Yaskawa INFORM job: N_R2_D54(P)(-165,-90).JBI

/JOB
//NAME N_R2_D54(P)(-165,-90)
//POS
///NPOS 418,418,418,21,0,0
///TOOL 0
///POSTYPE PULSE
///PULSE
C00000=-39723,-76225,-106677,19950,71807,76871
C00001=-136716,-73683,-105524,19345,72156,77265
C00002=-161407,-91524,-110310,15012,103390,71507
C00003=-159933,-105942,-63343,4894,72862,63752
C00004=-161158,-104529,-58514,4950,70696,63247
C00005=-161668,-103884,-56534,4974,69842,63039
C00006=-161778,-102512,-54221,4996,69133,62972
C00007=-161760,-102726,-54587,4993,69247,62982
C00008=-161816,-102665,-54558,4992,69263,62964
C00009=-163044,-104500,-55207,5003,68794,62527
C00010=-161816,-102665,-54558,4992,69263,62964
C00011=-161303,-103338,-56557,4967,70114,63174
C00012=-160072,-104820,-61433,4909,72274,63681
C00013=-171279,-139675,-91122,7314,74940,61433
C00014=-160786,-120191,-86572,7704,81092,65337
C00015=-161517,-119982,-82352,7740,78693,64939
C00016=-161824,-119782,-80612,7757,77762,64776
C00017=-161934,-118571,-78477,7774,77087,64696
C00018=-161898,-118737,-78823,7771,77210,64716
C00019=-161973,-118676,-78783,7769,77224,64692
C00020=-163205,-120940,-79512,7761,76632,64235
C00021=-161973,-118676,-78783,7769,77224,64692
C00022=-161664,-118910,-80540,7751,78148,64855
C00023=-160927,-119214,-84804,7712,80524,65254
C00024=-170669,-154499,-108862,8582,79492,59623
C00025=-160866,-130175,-103256,9154,87324,63496
C00026=-161601,-130979,-99438,9146,84678,63052
C00027=-161908,-131130,-97845,9147,83668,62873
C00028=-162018,-130031,-95808,9153,82999,62786
C00029=-162011,-130213,-96119,9152,83096,62795
C00030=-162089,-130094,-96081,9149,83142,62772
C00031=-163326,-132893,-96929,9116,82375,62294
C00032=-162089,-130094,-96081,9149,83142,62772
C00033=-161779,-129993,-97692,9146,84137,62951
C00034=-161038,-129333,-101562,9150,86742,63395
C00035=-164208,-146274,-116147,-5663,80658,78475
C00036=-172457,-131111,-102504,-10822,75194,76159
C00037=-174484,-130450,-98260,-10690,72692,75663
C00038=-175320,-130052,-96514,-10635,71726,75451
C00039=-175466,-128922,-94464,-10657,71037,75460
C00040=-175415,-129062,-94788,-10656,71169,75467
C00041=-175494,-129100,-94788,-10647,71140,75441
C00042=-177063,-131522,-95540,-10496,70167,74966
C00043=-175494,-129100,-94788,-10647,71140,75441
C00044=-174655,-129535,-96550,-10701,72096,75655
C00045=-172620,-130306,-100836,-10831,74570,76157
C00046=-185476,-152836,-107470,-9889,65575,72355
C00047=-172370,-120582,-85424,-11113,70194,76647
C00048=-174396,-119219,-80852,-11015,67845,76138
C00049=-175231,-118580,-78981,-10974,66925,75923
C00050=-175377,-117338,-76830,-11009,66232,75936
C00051=-175358,-117539,-77175,-11003,66341,75932
C00052=-175389,-117510,-77167,-10998,66348,75920
C00053=-176957,-119476,-77818,-10848,65543,75427
C00054=-175389,-117510,-77167,-10998,66348,75920
C00055=-174552,-118176,-79054,-11039,67264,76137
C00056=-172519,-119613,-83665,-11134,69599,76649
C00057=-182787,-134787,-88740,-10457,63687,73508
C00058=-171653,-105129,-60487,-14223,60495,76409
C00059=-174094,-102685,-55336,-14102,58231,75776
C00060=-175092,-101639,-53233,-14049,57333,75512
C00061=-175238,-100225,-50886,-14136,56611,75552
C00062=-175227,-100493,-51313,-14118,56735,75540
C00063=-175234,-100467,-51279,-14118,56726,75538
C00064=-176798,-102054,-51863,-13921,56030,75027
C00065=-175234,-100467,-51279,-14118,56726,75538
C00066=-174232,-101534,-53401,-14169,57626,75804
C00067=-171784,-104034,-58596,-14285,59890,76439
C00068=-145436,-132678,-96384,-390,75100,72869
C00069=-145436,-153477,-122592,-390,33068,72869
C00070=-145436,-153477,-122592,-390,33068,72869
C00071=-145875,-137223,-99163,-150,44123,76557
C00072=-145875,-137223,-99163,3185,26782,75636
C00073=-145939,-91194,-32923,8725,9743,73059
C00074=-160530,-30732,15414,32644,16120,44715
C00075=-161197,-23323,24436,37351,14921,42434
C00076=-161451,-20239,28250,39583,14417,41366
C00077=-161567,-18480,31613,42866,13575,39840
C00078=-161451,-20239,28250,39583,14417,41366
C00079=-161554,-18653,31308,42567,13643,39979
C00080=-160680,-16153,33400,41106,13277,40797
C00081=-161554,-18653,31308,42567,13643,39979
C00082=-161301,-21808,27395,40043,14138,41179
C00083=-160636,-29361,18168,34773,15327,43713
C00084=-135097,-31981,12391,41808,21062,54767
C00085=-134676,-25064,21391,45092,19411,53273
C00086=-134515,-22180,25183,46702,18734,52540
C00087=-134549,-20535,28420,49316,17967,51307
C00088=-134515,-22180,25183,46702,18734,52540
C00089=-134524,-20794,27979,48970,18047,51474
C00090=-134216,-18019,30231,48569,17928,51714
C00091=-134524,-20794,27979,48970,18047,51474
C00092=-134686,-23744,24097,47169,18719,52292
C00093=-135108,-30798,14911,43514,20363,53953
C00094=-130481,-37639,8518,34399,19575,58835
C00095=-121039,-28855,19333,23036,15252,65666
C00096=-121011,-21578,28921,26549,13273,64058
C00097=-121000,-18515,32998,28417,12436,63207
C00098=-120993,-15389,35919,28821,12265,63024
C00099=-120992,-16231,35105,28668,12325,63094
C00100=-120955,-16185,35150,28595,12310,63133
C00101=-120947,-14803,38264,31475,11256,61826
C00102=-120955,-16185,35150,28595,12310,63133
C00103=-120965,-19293,30991,26642,13171,64023
C00104=-120992,-26652,21234,23002,15205,65690
C00105=-121034,-28864,19164,22885,15343,65737
C00106=-121006,-21600,28739,26348,13362,64150
C00107=-120995,-18542,32808,28186,12525,63313
C00108=-120988,-15417,35727,28583,12354,63133
C00109=-120987,-16270,34916,28447,12408,63195
C00110=-120960,-16276,34878,28343,12418,63248
C00111=-120951,-14903,37981,31166,11363,61965
C00112=-120960,-16276,34878,28343,12418,63248
C00113=-120970,-19376,30730,26427,13278,64121
C00114=-120997,-26718,20994,22848,15312,65760
C00115=-145944,-87260,-27117,10373,8213,72316
C00116=-145875,-137223,-99163,-150,44123,76557
C00117=-112511,-157780,-119223,2457,-6594,76654
C00118=11401,-148032,-125424,11666,7065,68213
C00119=142233,-149944,-129024,-911,-4518,68213
C00120=169505,-149944,-129024,-911,70958,68213
C00121=146394,-132104,-100968,-948,62860,68213
C00122=112791,-124617,-91952,-2798,37533,68213
C00123=106222,-89941,-31656,13671,10104,57260
C00124=82158,-48543,-2966,1325,13441,54823
C00125=80586,-41795,4396,5777,12442,52566
C00126=79993,-39043,7456,7682,12022,51612
C00127=79856,-37591,10346,8813,11012,51078
C00128=79993,-39043,7456,7682,12022,51612
C00129=79847,-37520,10196,8740,11140,51110
C00130=80816,-35190,11887,5696,11217,52637
C00131=79847,-37520,10196,8740,11140,51110
C00132=80282,-36294,10063,6975,11807,51976
C00133=78629,-35044,10826,11506,12150,49671
C00134=80282,-36294,10063,6975,11807,51976
C00135=80868,-39067,6944,5071,12260,52929
C00136=82418,-45851,-550,665,13335,55161
C00137=92120,-47547,-3880,43195,24282,57629
C00138=92989,-41258,4025,45082,22690,56839
C00139=93323,-38677,7308,46001,22040,56447
C00140=93231,-37263,10172,47990,21363,55477
C00141=93244,-37464,9766,47701,21458,55618
C00142=93217,-37472,9805,47776,21451,55577
C00143=93881,-34964,11606,46865,21260,56119
C00144=93217,-37472,9805,47776,21451,55577
C00145=92880,-40093,6467,46755,22101,56015
C00146=92004,-46469,-1557,44658,23694,56897
C00147=90954,-53679,-8836,41955,25313,57794
C00148=91826,-47850,-3297,40845,25075,58444
C00149=92665,-41617,4654,42646,23429,57689
C00150=92987,-39055,7956,43520,22755,57315
C00151=93637,-36349,10201,42940,22473,57699
C00152=93435,-37229,9459,43112,22566,57584
C00153=93452,-37176,9500,43093,22560,57595
C00154=93243,-36182,12056,45087,21878,56602
C00155=93452,-37176,9500,43093,22560,57595
C00156=93139,-39751,6161,42190,23244,57984
C00157=92328,-46007,-1869,40331,24912,58771
C00158=106053,-48274,-3679,24965,19911,68135
C00159=106490,-41909,4331,26396,18284,67524
C00160=106658,-39298,7657,27116,17602,67212
C00161=106992,-36485,9961,26547,17529,67529
C00162=106885,-37411,9220,26746,17543,67420
C00163=106858,-37280,9353,26808,17538,67387
C00164=106753,-36322,11886,28592,16620,66539
C00165=106858,-37280,9353,26808,17538,67387
C00166=106695,-39904,5987,26065,18235,67710
C00167=106272,-46291,-2109,24590,19898,68344
C00168=112789,-102321,-56983,-3686,27485,364
C00169=146400,-134057,-103996,-943,63719,0
C00170=169505,-149944,-129024,-911,70958,0
C00171=130655,-113723,-117082,25754,15756,-2874
C00172=135046,-120043,-103653,15284,86568,-5166
C00173=145615,-106362,-63187,-723,70163,-73293
C00174=146466,-105075,-58388,-761,67879,-72986
C00175=146823,-104478,-56420,-778,66977,-72857
C00176=146913,-103100,-54104,-785,66261,-72822
C00177=146896,-103321,-54481,-784,66380,-72828
C00178=146930,-103303,-54456,-785,66374,-72816
C00179=147752,-105301,-55146,-816,65779,-72529
C00180=146930,-103303,-54456,-785,66374,-72816
C00181=146572,-103927,-56444,-768,67273,-72946
C00182=145715,-105287,-61291,-729,69549,-73255
C00183=171650,-107140,-63446,-1518,70275,-64361
C00184=173287,-105427,-58518,-1584,68154,-63772
C00185=173966,-104665,-56500,-1612,67317,-63527
C00186=174133,-103244,-54172,-1624,66618,-63460
C00187=174102,-103467,-54542,-1622,66730,-63472
C00188=174124,-103459,-54528,-1623,66726,-63465
C00189=175690,-105095,-55115,-1671,66277,-62921
C00190=174124,-103459,-54528,-1623,66726,-63465
C00191=173441,-104247,-56565,-1594,67561,-63711
C00192=171797,-106025,-61539,-1527,69677,-64303
C00193=172067,-142516,-91927,-1579,69887,-64201
C00194=158554,-122099,-87128,-1107,76938,-68913
C00195=159816,-121469,-82765,-1155,74595,-68460
C00196=160342,-121108,-80972,-1176,73684,-68271
C00197=160473,-119858,-78826,-1184,73009,-68220
C00198=160428,-120039,-79193,-1181,73141,-68237
C00199=160498,-119927,-79132,-1183,73161,-68213
C00200=161713,-122217,-79858,-1224,72450,-67790
C00201=160498,-119927,-79132,-1183,73161,-68213
C00202=159970,-120317,-80940,-1163,74066,-68402
C00203=158703,-121030,-85342,-1113,76391,-68857
C00204=146314,-120813,-86096,-9127,79912,-67896
C00205=146622,-120599,-81858,-9192,77479,-67610
C00206=146752,-120400,-80110,-9222,76532,-67495
C00207=146842,-119169,-77966,-9246,75864,-67413
C00208=146820,-119364,-78331,-9241,75984,-67430
C00209=146885,-119278,-78275,-9240,76001,-67409
C00210=147707,-121738,-79048,-9257,75314,-67076
C00211=146885,-119278,-78275,-9240,76001,-67409
C00212=146754,-119512,-80039,-9209,76940,-67525
C00213=146440,-119819,-84321,-9140,79351,-67812
C00214=155523,-158038,-108692,-12028,78540,-59985
C00215=146278,-131003,-102442,-12197,86758,-63975
C00216=146586,-131732,-98581,-12215,84113,-63609
C00217=146715,-131858,-96973,-12228,83101,-63465
C00218=146805,-130721,-94921,-12239,82450,-63370
C00219=146785,-130904,-95271,-12237,82567,-63388
C00220=146849,-130807,-95220,-12234,82595,-63369
C00221=147671,-133832,-96117,-12221,81736,-63001
C00222=146849,-130807,-95220,-12234,82595,-63369
C00223=146718,-130727,-96846,-12219,83594,-63513
C00224=146405,-130133,-100757,-12196,86200,-63876
C00225=158544,-132803,-104138,-1091,81906,-68960
C00226=159807,-133058,-100141,-1135,79333,-68507
C00227=160333,-133001,-98484,-1154,78350,-68318
C00228=160464,-131842,-96431,-1160,77684,-68268
C00229=160451,-132065,-96789,-1159,77789,-68273
C00230=160492,-132058,-96770,-1161,77782,-68259
C00231=161711,-134907,-97617,-1200,76857,-67834
C00232=160492,-132058,-96770,-1161,77782,-68259
C00233=159962,-132161,-98446,-1141,78752,-68449
C00234=158692,-132041,-102492,-1096,81286,-68904
C00235=156826,-87942,-103937,-736,105721,-87489
C00236=169505,-149944,-129024,-911,70958,-83128
C00237=150507,-86641,-54293,519,90148,-72841
C00238=151369,-88103,-51157,670,87460,-72568
C00239=151736,-88579,-49833,735,86398,-72453
C00240=150989,-86589,-48973,604,86898,-72696
C00241=151671,-89413,-51514,724,87005,-72471
C00242=148082,-90121,-50394,94,85969,-73650
C00243=143132,-91840,-51004,-775,85441,-75265
C00244=146976,-90753,-50017,-4652,86696,-74785
C00245=146908,-90233,-51327,-4663,87762,-74847
C00246=146750,-88663,-54427,-4697,90459,-74999
C00247=138996,-91037,-55808,9599,86257,-77118
C00248=140471,-92130,-52470,9835,83504,-76839
C00249=141100,-92456,-51068,9940,82414,-76717
C00250=141053,-93334,-52762,9923,83002,-76685
C00251=140577,-90379,-50216,9857,83011,-76843
C00252=144996,-91269,-50653,10469,82289,-75432
C00253=149985,-89384,-49977,11106,82190,-73775
C00254=153573,-87749,-49376,11536,82166,-72575
C00255=152772,-87476,-50772,11420,83257,-72743
C00256=150878,-86516,-54099,11159,86009,-73133
C00257=149105,-124457,-82831,10826,84649,-69493
C00258=139000,-101106,-75137,9614,92835,-76611
C00259=140475,-103328,-72336,9790,89833,-76340
C00260=141104,-104075,-71142,9873,88654,-76219
C00261=141057,-104785,-72699,9868,89245,-76189
C00262=140580,-101654,-70216,9803,89383,-76340
C00263=145001,-102673,-70675,10394,88598,-74902
C00264=150000,-100447,-69914,11023,88607,-73199
C00265=153588,-98526,-69240,11447,88674,-71968
C00266=152788,-97837,-70424,11359,89848,-72134
C00267=150894,-95766,-73199,11169,92832,-72516
C00268=150552,-95295,-72399,-4699,99242,-66870
C00269=151413,-97894,-69811,-4477,96371,-66468
C00270=151780,-98798,-68699,-4388,95246,-66304
C00271=151033,-96513,-67772,-4550,95807,-66577
C00272=151715,-99450,-70241,-4408,95854,-66347
C00273=148132,-100598,-69327,-5140,94495,-67509
C00274=143063,-102657,-70026,-6167,93518,-69177
C00275=146947,-101738,-68785,-10036,94570,-68905
C00276=146881,-100809,-69898,-10076,95707,-69020
C00277=146724,-98150,-72488,-10195,98604,-69311
C00278=156406,-129769,-96261,-9576,101180,-59267
C00279=152479,-99924,-86311,-11084,109498,-61410
C00280=153216,-103934,-84323,-10652,106370,-60850
C00281=153530,-105367,-83436,-10489,105150,-60628
C00282=152748,-102760,-82415,-10743,105747,-60963
C00283=153463,-105818,-84866,-10546,105779,-60707
C00284=149940,-107591,-84196,-11408,104000,-61813
C00285=145065,-110118,-85037,-12614,102512,-63411
C00286=141170,-111760,-85570,-13543,101381,-64679
C00287=141083,-110376,-86518,-13642,102626,-64851
C00288=140879,-106472,-88660,-13928,105824,-65295
C00289=139012,-108324,-91751,9773,99260,-76104
C00290=140488,-112023,-89529,9880,95858,-75861
C00291=141117,-113312,-88549,9938,94534,-75749
C00292=141071,-113826,-89993,9945,95155,-75715
C00293=140593,-110413,-87497,9885,95428,-75859
C00294=145016,-111613,-88000,10463,94569,-74398
C00295=150011,-108930,-87112,11100,94719,-72653
C00296=153600,-106623,-86327,11531,94906,-71389
C00297=152799,-105405,-87291,11473,96215,-71546
C00298=150904,-101897,-89475,11366,99570,-71898
C00299=126224,-114648,-117374,36487,17100,-46505
C00300=161894,-128023,-129024,-3891,66929,0
C00301=169505,-149944,-129024,-911,70958,68213
C00302=146345,-116770,-77350,-998,56205,68213
C00303=107194,-71790,-14984,39783,21053,48304
C00304=107156,-65179,-7591,41825,20185,47324
C00305=107142,-62504,-4543,42769,19814,46874
C00306=106800,-64490,-5882,43466,19814,46482
C00307=107246,-63323,-6435,41303,20331,47588
C00308=70029,-46302,3349,53937,40189,34366
C00309=69578,-48817,175,53379,40826,34608
C00310=68404,-54960,-7486,52160,42404,35115
C00311=92169,-90677,-38321,17628,21409,69664
C00312=104331,-95917,-39395,-3234,13257,85275
C00313=104468,-89231,-32897,-3735,12700,85524
C00314=104519,-86574,-30246,-3950,12437,85630
C00315=104018,-88444,-31057,-2700,11957,84983
C00316=104716,-87040,-31804,-4240,13164,85793
C00317=67078,-70441,-24138,47983,28112,55943
C00318=72664,-72074,-22716,43378,19620,45867
C00319=72698,-74754,-25444,42764,19829,46163
C00320=72788,-81468,-32110,41462,20280,46794
C00321=111872,-135193,-95342,-2266,25761,38955
C00322=112791,-119013,-83053,-2974,34939,68213
C00323=146364,-125626,-92975,-983,57710,68213
C00324=169505,-149944,-129024,-911,70958,68213
C00325=133842,-149944,-129024,-911,13808,68213
C00326=90580,-158557,-127215,5410,7231,72011
C00327=12469,-167082,-125424,11666,-5656,75770
C00328=-137258,-84249,-120477,10166,64820,76481
C00329=-160540,-100856,-113062,23154,68828,67580
C00330=-177338,-94304,-53616,492,89079,62806
C00331=-179085,-95046,-50077,110,86527,62233
C00332=-179834,-95235,-48596,-53,85519,61993
C00333=-179722,-96248,-50353,-29,86079,62028
C00334=-178336,-93703,-47978,273,85923,62473
C00335=-176530,-97945,-49475,669,84655,63046
C00336=-171706,-101321,-50515,1726,83493,64567
C00337=-167741,-103665,-51199,2593,82611,65807
C00338=-167171,-103532,-52749,2712,83615,66008
C00339=-165860,-102931,-56466,2988,86164,66485
C00340=-166108,-127396,-81125,5974,94843,53127
C00341=-158272,-93134,-70047,8830,104781,56387
C00342=-159421,-95524,-67393,8374,102072,55789
C00343=-159910,-96349,-66257,8192,101010,55546
C00344=-159846,-97004,-67807,8231,101615,55609
C00345=-158998,-94211,-65368,8476,101463,55894
C00346=-156481,-98582,-67072,9157,100006,56663
C00347=-151660,-101260,-68022,10482,98647,58220
C00348=-147866,-103024,-68632,11496,97618,59434
C00349=-147574,-102225,-69820,11616,98696,59637
C00350=-146893,-99892,-72601,11929,101449,60141
C00351=-154176,-136144,-99393,7036,97628,61519
C00352=-152138,-100329,-87963,8214,108619,62918
C00353=-153017,-104433,-86004,7830,105423,62383
C00354=-153391,-105899,-85127,7682,104178,62169
C00355=-153339,-106312,-86540,7722,104825,62229
C00356=-152618,-103240,-84090,7904,104825,62487
C00357=-149803,-108157,-85918,8534,103150,63375
C00358=-144933,-110724,-86797,9658,101831,65000
C00359=-141045,-112392,-87358,10527,100841,66291
C00360=-140889,-110956,-88289,10621,102110,66456
C00361=-140527,-106910,-90384,10885,105374,66878
C00362=-148014,-100498,-99830,-10640,107359,74545
C00363=-152716,-92792,-83729,-23070,96978,80334
C00364=-154781,-96001,-81564,-23037,93647,80218
C00365=-155647,-97118,-80613,-23047,92334,80152
C00366=-154878,-94597,-79547,-23024,93139,80280
C00367=-155595,-97427,-81992,-23066,92985,80045
C00368=-158814,-94590,-79629,-23223,92083,79035
C00369=-162731,-91043,-78206,-23386,91848,77637
C00370=-165587,-88135,-77004,-23466,91731,76607
C00371=-164661,-87102,-77942,-23485,93015,76696
C00372=-162435,-84125,-80080,-23579,96268,76873
C00373=-158516,-112098,-90966,-23434,90383,79484
C00374=-151919,-102148,-74374,-18289,88823,80795
C00375=-153945,-103844,-71356,-18502,85775,80539
C00376=-154805,-104384,-70079,-18603,84572,80420
C00377=-153940,-102135,-69222,-18508,85363,80604
C00378=-154746,-105132,-71653,-18586,85141,80354
C00379=-158469,-102205,-69335,-18918,84371,79161
C00380=-163078,-99000,-68205,-19249,84210,77556
C00381=-166328,-96392,-67254,-19439,84163,76409
C00382=-165367,-95898,-68508,-19360,85359,76560
C00383=-163080,-94324,-71470,-19199,88386,76895
C00384=-168755,-117883,-78463,-23858,79273,80780
C00385=-162659,-103826,-55618,-25977,72070,81323
C00386=-166238,-103089,-51471,-26508,69052,80706
C00387=-167751,-102685,-49757,-26733,67841,80435
C00388=-166351,-100995,-49160,-26571,68707,80747
C00389=-167649,-103804,-51545,-26638,68343,80351
C00390=-171717,-100365,-49077,-26772,67352,79068
C00391=-176541,-97022,-48043,-26695,66876,77359
C00392=-179845,-94338,-47169,-26559,66637,76157
C00393=-178363,-94810,-48879,-26415,67811,76439
C00394=-174798,-95723,-53014,-26065,70755,77095
C00395=-137258,-84249,-120477,10166,64820,0
C00396=-145436,-153477,-122592,-390,33068,0
C00397=-145436,-153477,-122592,-390,33068,0
C00398=-145875,-137223,-99163,-150,44123,0
C00399=-84324,-58786,-9259,-66850,52098,-39426
C00400=-87232,-53748,-2579,-68318,49731,-39064
C00401=-88364,-51659,185,-68961,48807,-38888
C00402=-87658,-53409,-905,-69052,49144,-38654
C00403=-88659,-52210,-1515,-68378,48926,-39360
C00404=-128534,-57912,-2626,-72555,23972,-44877
C00405=-127801,-60507,-5562,-71635,24574,-45197
C00406=-125863,-66894,-12673,-69713,26136,-45808
C00407=-123683,-86538,-29853,-33918,27431,-1450
C00408=-121135,-57598,-3033,2619,26844,48411
C00409=-121118,-57251,-2489,2618,26687,48415
C00410=-121111,-57244,-2487,2611,26689,48420
C00411=-121122,-59280,-3914,2636,26521,48406
C00412=-121119,-58008,-4354,2552,27445,48448
C00413=-121112,-57255,-2369,2619,26611,48416
C00414=-121119,-57262,-2372,2625,26609,48412
C00415=-121135,-57547,-2815,2630,26736,48406
C00416=-145875,-137223,-99163,-150,44123,0
C00417=-39723,-76225,-106677,19950,71807,76871
BC00000=295325,674563,1075175
BC00001=353535,895977,1075175
BC00002=353535,975867,1075175
BC00003=331218,1039193,1075175
BC00004=331218,1039193,1075175
BC00005=331218,1039193,1075175
BC00006=331218,1039193,1075175
BC00007=331218,1039193,1075175
BC00008=331218,1039193,1075175
BC00009=331218,1039193,1075175
BC00010=331218,1039193,1075175
BC00011=331218,1039193,1075175
BC00012=331218,1039193,1075175
BC00013=324452,1071332,1075175
BC00014=324452,1071332,1075175
BC00015=324452,1071332,1075175
BC00016=324452,1071332,1075175
BC00017=324452,1071332,1075175
BC00018=324452,1071332,1075175
BC00019=324452,1071332,1075175
BC00020=324452,1071332,1075175
BC00021=324452,1071332,1075175
BC00022=324452,1071332,1075175
BC00023=324452,1071332,1075175
BC00024=321407,1100758,1075175
BC00025=321407,1100758,1075175
BC00026=321407,1100758,1075175
BC00027=321407,1100758,1075175
BC00028=321407,1100758,1075175
BC00029=321407,1100758,1075175
BC00030=321407,1100758,1075175
BC00031=321407,1100758,1075175
BC00032=321407,1100758,1075175
BC00033=321407,1100758,1075175
BC00034=321407,1100758,1075175
BC00035=308537,1111089,1075175
BC00036=308537,1111089,1075175
BC00037=308537,1111089,1075175
BC00038=308537,1111089,1075175
BC00039=308537,1111089,1075175
BC00040=308537,1111089,1075175
BC00041=308537,1111089,1075175
BC00042=308537,1111089,1075175
BC00043=308537,1111089,1075175
BC00044=308537,1111089,1075175
BC00045=308537,1111089,1075175
BC00046=308537,1111089,1075175
BC00047=308670,1082030,1075175
BC00048=308670,1082030,1075175
BC00049=308670,1082030,1075175
BC00050=308670,1082030,1075175
BC00051=308670,1082030,1075175
BC00052=308670,1082030,1075175
BC00053=308670,1082030,1075175
BC00054=308670,1082030,1075175
BC00055=308670,1082030,1075175
BC00056=308670,1082030,1075175
BC00057=308670,1082030,1075175
BC00058=315403,1047567,1075175
BC00059=315403,1047567,1075175
BC00060=315403,1047567,1075175
BC00061=315403,1047567,1075175
BC00062=315403,1047567,1075175
BC00063=315403,1047567,1075175
BC00064=315403,1047567,1075175
BC00065=315403,1047567,1075175
BC00066=315403,1047567,1075175
BC00067=315403,1047567,1075175
BC00068=334035,1006363,1075175
BC00069=334035,960963,1075175
BC00070=369533,796939,1075175
BC00071=369533,796939,1075175
BC00072=324907,880615,715339
BC00073=299333,903943,1016574
BC00074=320965,885240,1075175
BC00075=320965,885240,1075175
BC00076=320965,885240,1075175
BC00077=320965,885240,1075175
BC00078=320965,885240,1075175
BC00079=320965,885240,1075175
BC00080=320965,885240,1075175
BC00081=320965,885240,1075175
BC00082=320965,885240,1075175
BC00083=320965,885240,1075175
BC00084=287794,865868,1075175
BC00085=287794,865868,1075175
BC00086=287794,865868,1075175
BC00087=287794,865868,1075175
BC00088=287794,865868,1075175
BC00089=287794,865868,1075175
BC00090=287794,865868,1075175
BC00091=287794,865868,1075175
BC00092=287794,865868,1075175
BC00093=287794,865868,1075175
BC00094=279992,861447,1075175
BC00095=264389,852604,1075175
BC00096=264389,852604,1075175
BC00097=264389,852604,1075175
BC00098=264389,852604,1075175
BC00099=264389,852604,1075175
BC00100=264389,852604,1075175
BC00101=264389,852604,1075175
BC00102=264389,852604,1075175
BC00103=264389,852604,1075175
BC00104=264389,852604,1075175
BC00105=317167,852667,1075175
BC00106=317167,852667,1075175
BC00107=317167,852667,1075175
BC00108=317167,852667,1075175
BC00109=317167,852667,1075175
BC00110=317167,852667,1075175
BC00111=317167,852667,1075175
BC00112=317167,852667,1075175
BC00113=317167,852667,1075175
BC00114=317167,852667,1075175
BC00115=324907,880615,1043823
BC00116=369533,796939,1075175
BC00117=372496,892269,1075175
BC00118=398190,1030285,1075175
BC00119=387158,1273206,1073754
BC00120=387158,1273206,1073754
BC00121=354276,1245348,919518
BC00122=302489,1244324,830763
BC00123=299772,1224612,1018067
BC00124=266448,1223446,1015899
BC00125=266448,1223446,1015899
BC00126=266448,1223446,1015899
BC00127=266448,1223446,1015899
BC00128=266448,1223446,1015899
BC00129=266448,1223446,1015899
BC00130=266448,1223446,1015899
BC00131=266448,1223446,1015899
BC00132=266448,1223446,1015899
BC00133=266448,1223446,1015899
BC00134=266448,1223446,1015899
BC00135=266448,1223446,1015899
BC00136=266448,1223446,1015899
BC00137=284185,1241172,1035391
BC00138=284185,1241172,1035391
BC00139=284185,1241172,1035391
BC00140=284185,1241172,1035391
BC00141=284185,1241172,1035391
BC00142=284185,1241172,1035391
BC00143=284185,1241172,1035391
BC00144=284185,1241172,1035391
BC00145=284185,1241172,1035391
BC00146=284185,1241172,1035391
BC00147=283221,1247342,1023689
BC00148=282418,1252484,1013938
BC00149=282418,1252484,1013938
BC00150=282418,1252484,1013938
BC00151=282418,1252484,1013938
BC00152=282418,1252484,1013938
BC00153=282418,1252484,1013938
BC00154=282418,1252484,1013938
BC00155=282418,1252484,1013938
BC00156=282418,1252484,1013938
BC00157=282418,1252484,1013938
BC00158=251392,1257834,1013840
BC00159=251392,1257834,1013840
BC00160=251392,1257834,1013840
BC00161=251392,1257834,1013840
BC00162=251392,1257834,1013840
BC00163=251392,1257834,1013840
BC00164=251392,1257834,1013840
BC00165=251392,1257834,1013840
BC00166=251392,1257834,1013840
BC00167=251392,1257834,1013840
BC00168=302489,1244324,999744
BC00169=354276,1245348,903959
BC00170=387158,1273206,1073754
BC00171=343908,1138057,1075175
BC00172=340753,1115300,1075175
BC00173=324450,1090582,1075175
BC00174=324450,1090582,1075175
BC00175=324450,1090582,1075175
BC00176=324450,1090582,1075175
BC00177=324450,1090582,1075175
BC00178=324450,1090582,1075175
BC00179=324450,1090582,1075175
BC00180=324450,1090582,1075175
BC00181=324450,1090582,1075175
BC00182=324450,1090582,1075175
BC00183=316029,1077484,1075175
BC00184=316029,1077484,1075175
BC00185=316029,1077484,1075175
BC00186=316029,1077484,1075175
BC00187=316029,1077484,1075175
BC00188=316029,1077484,1075175
BC00189=316029,1077484,1075175
BC00190=316029,1077484,1075175
BC00191=316029,1077484,1075175
BC00192=316029,1077484,1075175
BC00193=304893,1052205,1075175
BC00194=304893,1052205,1075175
BC00195=304893,1052205,1075175
BC00196=304893,1052205,1075175
BC00197=304893,1052205,1075175
BC00198=304893,1052205,1075175
BC00199=304893,1052205,1075175
BC00200=304893,1052205,1075175
BC00201=304893,1052205,1075175
BC00202=304893,1052205,1075175
BC00203=304893,1052205,1075175
BC00204=308849,1057402,1075175
BC00205=308849,1057402,1075175
BC00206=308849,1057402,1075175
BC00207=308849,1057402,1075175
BC00208=308849,1057402,1075175
BC00209=308849,1057402,1075175
BC00210=308849,1057402,1075175
BC00211=308849,1057402,1075175
BC00212=308849,1057402,1075175
BC00213=308849,1057402,1075175
BC00214=303096,1026670,1075175
BC00215=303096,1026670,1075175
BC00216=303096,1026670,1075175
BC00217=303096,1026670,1075175
BC00218=303096,1026670,1075175
BC00219=303096,1026670,1075175
BC00220=303096,1026670,1075175
BC00221=303096,1026670,1075175
BC00222=303096,1026670,1075175
BC00223=303096,1026670,1075175
BC00224=303096,1026670,1075175
BC00225=304929,1022999,1075175
BC00226=304929,1022999,1075175
BC00227=304929,1022999,1075175
BC00228=304929,1022999,1075175
BC00229=304929,1022999,1075175
BC00230=304929,1022999,1075175
BC00231=304929,1022999,1075175
BC00232=304929,1022999,1075175
BC00233=304929,1022999,1075175
BC00234=304929,1022999,1075175
BC00235=340054,1089258,1073754
BC00236=340054,1089258,1073754
BC00237=318456,1078545,1057631
BC00238=318456,1078545,1057631
BC00239=318456,1078545,1057631
BC00240=318456,1078545,1057631
BC00241=318456,1078545,1057631
BC00242=318456,1078545,1057631
BC00243=318456,1078545,1057631
BC00244=318456,1078545,1057631
BC00245=318456,1078545,1057631
BC00246=318456,1078545,1057631
BC00247=310811,1078391,1057817
BC00248=310811,1078391,1057817
BC00249=310811,1078391,1057817
BC00250=310811,1078391,1057817
BC00251=310811,1078391,1057817
BC00252=310811,1078391,1057817
BC00253=310811,1078391,1057817
BC00254=310811,1078391,1057817
BC00255=310811,1078391,1057817
BC00256=310811,1078391,1057817
BC00257=314509,1043182,1075175
BC00258=310928,1045787,1075175
BC00259=310928,1045787,1075175
BC00260=310928,1045787,1075175
BC00261=310928,1045787,1075175
BC00262=310928,1045787,1075175
BC00263=310928,1045787,1075175
BC00264=310928,1045787,1075175
BC00265=310928,1045787,1075175
BC00266=310928,1045787,1075175
BC00267=310928,1045787,1075175
BC00268=309679,1045444,1075175
BC00269=309679,1045444,1075175
BC00270=309679,1045444,1075175
BC00271=309679,1045444,1075175
BC00272=309679,1045444,1075175
BC00273=309679,1045444,1075175
BC00274=309679,1045444,1075175
BC00275=309679,1045444,1075175
BC00276=309679,1045444,1075175
BC00277=309679,1045444,1075175
BC00278=293203,1011474,1075175
BC00279=300031,1014156,1075175
BC00280=300031,1014156,1075175
BC00281=300031,1014156,1075175
BC00282=300031,1014156,1075175
BC00283=300031,1014156,1075175
BC00284=300031,1014156,1075175
BC00285=300031,1014156,1075175
BC00286=300031,1014156,1075175
BC00287=300031,1014156,1075175
BC00288=300031,1014156,1075175
BC00289=311027,1016676,1075175
BC00290=311027,1016676,1075175
BC00291=311027,1016676,1075175
BC00292=311027,1016676,1075175
BC00293=311027,1016676,1075175
BC00294=311027,1016676,1075175
BC00295=311027,1016676,1075175
BC00296=311027,1016676,1075175
BC00297=311027,1016676,1075175
BC00298=311027,1016676,1075175
BC00299=312632,1138057,1075175
BC00300=363646,1230569,1074202
BC00301=387158,1273206,1073754
BC00302=354276,1245348,1037481
BC00303=264611,1222880,1007534
BC00304=264611,1222880,1007534
BC00305=264611,1222880,1007534
BC00306=264611,1222880,1007534
BC00307=264611,1222880,1007534
BC00308=264611,1222880,1007534
BC00309=264611,1222880,1007534
BC00310=264611,1222880,1007534
BC00311=281404,1203194,953762
BC00312=292031,1197764,938171
BC00313=292031,1197764,938171
BC00314=292031,1197764,938171
BC00315=292031,1197764,938171
BC00316=292031,1197764,938171
BC00317=292031,1197764,938171
BC00318=292031,1197764,938171
BC00319=292031,1197764,938171
BC00320=292031,1197764,938171
BC00321=305225,1224612,728593
BC00322=302489,1244324,875371
BC00323=354276,1245348,995177
BC00324=387158,1273206,1073754
BC00325=387158,1273206,1073754
BC00326=392702,1151116,1074468
BC00327=398190,1030285,1075175
BC00328=353817,923990,1075175
BC00329=381896,966588,1075175
BC00330=325812,1070585,1075175
BC00331=325812,1070585,1075175
BC00332=325812,1070585,1075175
BC00333=325812,1070585,1075175
BC00334=325812,1070585,1075175
BC00335=325812,1070585,1075175
BC00336=325812,1070585,1075175
BC00337=325812,1070585,1075175
BC00338=325812,1070585,1075175
BC00339=325812,1070585,1075175
BC00340=298621,1092729,1075175
BC00341=306802,1084796,1075175
BC00342=306802,1084796,1075175
BC00343=306802,1084796,1075175
BC00344=306802,1084796,1075175
BC00345=306802,1084796,1075175
BC00346=306802,1084796,1075175
BC00347=306802,1084796,1075175
BC00348=306802,1084796,1075175
BC00349=306802,1084796,1075175
BC00350=306802,1084796,1075175
BC00351=296440,1116752,1075175
BC00352=304452,1108725,1075175
BC00353=304452,1108725,1075175
BC00354=304452,1108725,1075175
BC00355=304452,1108725,1075175
BC00356=304452,1108725,1075175
BC00357=304452,1108725,1075175
BC00358=304452,1108725,1075175
BC00359=304452,1108725,1075175
BC00360=304452,1108725,1075175
BC00361=304452,1108725,1075175
BC00362=314166,1107968,1075175
BC00363=318465,1104321,1075175
BC00364=318465,1104321,1075175
BC00365=318465,1104321,1075175
BC00366=318465,1104321,1075175
BC00367=318465,1104321,1075175
BC00368=318465,1104321,1075175
BC00369=318465,1104321,1075175
BC00370=318465,1104321,1075175
BC00371=318465,1104321,1075175
BC00372=318465,1104321,1075175
BC00373=319691,1106269,1075175
BC00374=303635,1086463,1075175
BC00375=303635,1086463,1075175
BC00376=303635,1086463,1075175
BC00377=303635,1086463,1075175
BC00378=303635,1086463,1075175
BC00379=303635,1086463,1075175
BC00380=303635,1086463,1075175
BC00381=303635,1086463,1075175
BC00382=303635,1086463,1075175
BC00383=303635,1086463,1075175
BC00384=318817,1096650,1075175
BC00385=319676,1072931,1065034
BC00386=319676,1072931,1065034
BC00387=319676,1072931,1065034
BC00388=319676,1072931,1065034
BC00389=319676,1072931,1065034
BC00390=319676,1072931,1065034
BC00391=319676,1072931,1065034
BC00392=319676,1072931,1065034
BC00393=319676,1072931,1065034
BC00394=319676,1072931,1065034
BC00395=353817,923990,1075175
BC00396=334035,960963,1075175
BC00397=369533,796939,1075175
BC00398=369533,796939,1075175
BC00399=279256,911928,995377
BC00400=279256,911928,995377
BC00401=279256,911928,995377
BC00402=279256,911928,995377
BC00403=279256,911928,995377
BC00404=279256,911928,995377
BC00405=279256,911928,995377
BC00406=279256,911928,995377
BC00407=306660,907064,1033541
BC00408=336555,901758,1075175
BC00409=333838,905015,1054565
BC00410=332752,906318,1045544
BC00411=332752,906318,1045544
BC00412=332752,906318,1045544
BC00413=278810,906221,1045178
BC00414=279896,904918,1054199
BC00415=282613,901661,1075175
BC00416=369533,796939,1075175
BC00417=295325,674563,1075175
EC00000=-1463287,-556475
EC00001=-1463287,-556475
EC00002=-1463287,-556475
EC00003=-1463287,-556475
EC00004=-1463287,-556475
EC00005=-1463287,-556475
EC00006=-1463287,-556475
EC00007=-1463287,-556475
EC00008=-1463287,-556475
EC00009=-1463287,-556475
EC00010=-1463287,-556475
EC00011=-1463287,-556475
EC00012=-1463287,-556475
EC00013=-1463287,-556475
EC00014=-1463287,-556475
EC00015=-1463287,-556475
EC00016=-1463287,-556475
EC00017=-1463287,-556475
EC00018=-1463287,-556475
EC00019=-1463287,-556475
EC00020=-1463287,-556475
EC00021=-1463287,-556475
EC00022=-1463287,-556475
EC00023=-1463287,-556475
EC00024=-1463287,-556475
EC00025=-1463287,-556475
EC00026=-1463287,-556475
EC00027=-1463287,-556475
EC00028=-1463287,-556475
EC00029=-1463287,-556475
EC00030=-1463287,-556475
EC00031=-1463287,-556475
EC00032=-1463287,-556475
EC00033=-1463287,-556475
EC00034=-1463287,-556475
EC00035=-1463287,-556475
EC00036=-1463287,-556475
EC00037=-1463287,-556475
EC00038=-1463287,-556475
EC00039=-1463287,-556475
EC00040=-1463287,-556475
EC00041=-1463287,-556475
EC00042=-1463287,-556475
EC00043=-1463287,-556475
EC00044=-1463287,-556475
EC00045=-1463287,-556475
EC00046=-1463287,-556475
EC00047=-1463287,-556475
EC00048=-1463287,-556475
EC00049=-1463287,-556475
EC00050=-1463287,-556475
EC00051=-1463287,-556475
EC00052=-1463287,-556475
EC00053=-1463287,-556475
EC00054=-1463287,-556475
EC00055=-1463287,-556475
EC00056=-1463287,-556475
EC00057=-1463287,-556475
EC00058=-1463287,-556475
EC00059=-1463287,-556475
EC00060=-1463287,-556475
EC00061=-1463287,-556475
EC00062=-1463287,-556475
EC00063=-1463287,-556475
EC00064=-1463287,-556475
EC00065=-1463287,-556475
EC00066=-1463287,-556475
EC00067=-1463287,-556475
EC00068=-1463287,-556475
EC00069=-1463287,-556475
EC00070=-1463287,-556475
EC00071=-1463287,-556475
EC00072=-1463287,-556475
EC00073=-1463287,-556475
EC00074=-1463287,-556475
EC00075=-1463287,-556475
EC00076=-1463287,-556475
EC00077=-1463287,-556475
EC00078=-1463287,-556475
EC00079=-1463287,-556475
EC00080=-1463287,-556475
EC00081=-1463287,-556475
EC00082=-1463287,-556475
EC00083=-1463287,-556475
EC00084=-1463287,-556475
EC00085=-1463287,-556475
EC00086=-1463287,-556475
EC00087=-1463287,-556475
EC00088=-1463287,-556475
EC00089=-1463287,-556475
EC00090=-1463287,-556475
EC00091=-1463287,-556475
EC00092=-1463287,-556475
EC00093=-1463287,-556475
EC00094=-1463287,-556475
EC00095=-1463287,-556475
EC00096=-1463287,-556475
EC00097=-1463287,-556475
EC00098=-1463287,-556475
EC00099=-1463287,-556475
EC00100=-1463287,-556475
EC00101=-1463287,-556475
EC00102=-1463287,-556475
EC00103=-1463287,-556475
EC00104=-1463287,-556475
EC00105=-1463287,-556475
EC00106=-1463287,-556475
EC00107=-1463287,-556475
EC00108=-1463287,-556475
EC00109=-1463287,-556475
EC00110=-1463287,-556475
EC00111=-1463287,-556475
EC00112=-1463287,-556475
EC00113=-1463287,-556475
EC00114=-1463287,-556475
EC00115=-1463287,-556475
EC00116=-1463287,-556475
EC00117=-1463287,-556475
EC00118=-1595090,-3837
EC00119=-1729339,556475
EC00120=-1729339,556475
EC00121=-1729339,556475
EC00122=-1729339,556475
EC00123=-1729339,556475
EC00124=-1729339,556475
EC00125=-1729339,556475
EC00126=-1729339,556475
EC00127=-1729339,556475
EC00128=-1729339,556475
EC00129=-1729339,556475
EC00130=-1729339,556475
EC00131=-1729339,556475
EC00132=-1729339,556475
EC00133=-1729339,556475
EC00134=-1729339,556475
EC00135=-1729339,556475
EC00136=-1729339,556475
EC00137=-1729339,556475
EC00138=-1729339,556475
EC00139=-1729339,556475
EC00140=-1729339,556475
EC00141=-1729339,556475
EC00142=-1729339,556475
EC00143=-1729339,556475
EC00144=-1729339,556475
EC00145=-1729339,556475
EC00146=-1729339,556475
EC00147=-1729339,556475
EC00148=-1729339,556475
EC00149=-1729339,556475
EC00150=-1729339,556475
EC00151=-1729339,556475
EC00152=-1729339,556475
EC00153=-1729339,556475
EC00154=-1729339,556475
EC00155=-1729339,556475
EC00156=-1729339,556475
EC00157=-1729339,556475
EC00158=-1729339,556475
EC00159=-1729339,556475
EC00160=-1729339,556475
EC00161=-1729339,556475
EC00162=-1729339,556475
EC00163=-1729339,556475
EC00164=-1729339,556475
EC00165=-1729339,556475
EC00166=-1729339,556475
EC00167=-1729339,556475
EC00168=-1729339,556475
EC00169=-1729339,556475
EC00170=-1729339,556475
EC00171=-1729339,556475
EC00172=-1729339,556475
EC00173=-1729339,556475
EC00174=-1729339,556475
EC00175=-1729339,556475
EC00176=-1729339,556475
EC00177=-1729339,556475
EC00178=-1729339,556475
EC00179=-1729339,556475
EC00180=-1729339,556475
EC00181=-1729339,556475
EC00182=-1729339,556475
EC00183=-1729339,556475
EC00184=-1729339,556475
EC00185=-1729339,556475
EC00186=-1729339,556475
EC00187=-1729339,556475
EC00188=-1729339,556475
EC00189=-1729339,556475
EC00190=-1729339,556475
EC00191=-1729339,556475
EC00192=-1729339,556475
EC00193=-1729339,556475
EC00194=-1729339,556475
EC00195=-1729339,556475
EC00196=-1729339,556475
EC00197=-1729339,556475
EC00198=-1729339,556475
EC00199=-1729339,556475
EC00200=-1729339,556475
EC00201=-1729339,556475
EC00202=-1729339,556475
EC00203=-1729339,556475
EC00204=-1729339,556475
EC00205=-1729339,556475
EC00206=-1729339,556475
EC00207=-1729339,556475
EC00208=-1729339,556475
EC00209=-1729339,556475
EC00210=-1729339,556475
EC00211=-1729339,556475
EC00212=-1729339,556475
EC00213=-1729339,556475
EC00214=-1729339,556475
EC00215=-1729339,556475
EC00216=-1729339,556475
EC00217=-1729339,556475
EC00218=-1729339,556475
EC00219=-1729339,556475
EC00220=-1729339,556475
EC00221=-1729339,556475
EC00222=-1729339,556475
EC00223=-1729339,556475
EC00224=-1729339,556475
EC00225=-1729339,556475
EC00226=-1729339,556475
EC00227=-1729339,556475
EC00228=-1729339,556475
EC00229=-1729339,556475
EC00230=-1729339,556475
EC00231=-1729339,556475
EC00232=-1729339,556475
EC00233=-1729339,556475
EC00234=-1729339,556475
EC00235=-1729339,556475
EC00236=-1729339,556475
EC00237=-1729339,556475
EC00238=-1729339,556475
EC00239=-1729339,556475
EC00240=-1729339,556475
EC00241=-1729339,556475
EC00242=-1729339,556475
EC00243=-1729339,556475
EC00244=-1729339,556475
EC00245=-1729339,556475
EC00246=-1729339,556475
EC00247=-1729339,556475
EC00248=-1729339,556475
EC00249=-1729339,556475
EC00250=-1729339,556475
EC00251=-1729339,556475
EC00252=-1729339,556475
EC00253=-1729339,556475
EC00254=-1729339,556475
EC00255=-1729339,556475
EC00256=-1729339,556475
EC00257=-1729339,556475
EC00258=-1729339,556475
EC00259=-1729339,556475
EC00260=-1729339,556475
EC00261=-1729339,556475
EC00262=-1729339,556475
EC00263=-1729339,556475
EC00264=-1729339,556475
EC00265=-1729339,556475
EC00266=-1729339,556475
EC00267=-1729339,556475
EC00268=-1729339,556475
EC00269=-1729339,556475
EC00270=-1729339,556475
EC00271=-1729339,556475
EC00272=-1729339,556475
EC00273=-1729339,556475
EC00274=-1729339,556475
EC00275=-1729339,556475
EC00276=-1729339,556475
EC00277=-1729339,556475
EC00278=-1729339,556475
EC00279=-1729339,556475
EC00280=-1729339,556475
EC00281=-1729339,556475
EC00282=-1729339,556475
EC00283=-1729339,556475
EC00284=-1729339,556475
EC00285=-1729339,556475
EC00286=-1729339,556475
EC00287=-1729339,556475
EC00288=-1729339,556475
EC00289=-1729339,556475
EC00290=-1729339,556475
EC00291=-1729339,556475
EC00292=-1729339,556475
EC00293=-1729339,556475
EC00294=-1729339,556475
EC00295=-1729339,556475
EC00296=-1729339,556475
EC00297=-1729339,556475
EC00298=-1729339,556475
EC00299=-1729339,556475
EC00300=-1729339,556475
EC00301=-1729339,556475
EC00302=-1729339,556475
EC00303=-1729339,556475
EC00304=-1729339,556475
EC00305=-1729339,556475
EC00306=-1729339,556475
EC00307=-1729339,556475
EC00308=-1729339,556475
EC00309=-1729339,556475
EC00310=-1729339,556475
EC00311=-1729339,556475
EC00312=-1729339,556475
EC00313=-1729339,556475
EC00314=-1729339,556475
EC00315=-1729339,556475
EC00316=-1729339,556475
EC00317=-1729339,556475
EC00318=-1729339,556475
EC00319=-1729339,556475
EC00320=-1729339,556475
EC00321=-1729339,556475
EC00322=-1729339,556475
EC00323=-1729339,556475
EC00324=-1729339,556475
EC00325=-1729339,556475
EC00326=-1661867,274867
EC00327=-1595090,-3837
EC00328=-1463287,-556475
EC00329=-1463287,-556475
EC00330=-1463287,-556475
EC00331=-1463287,-556475
EC00332=-1463287,-556475
EC00333=-1463287,-556475
EC00334=-1463287,-556475
EC00335=-1463287,-556475
EC00336=-1463287,-556475
EC00337=-1463287,-556475
EC00338=-1463287,-556475
EC00339=-1463287,-556475
EC00340=-1463287,-556475
EC00341=-1463287,-556475
EC00342=-1463287,-556475
EC00343=-1463287,-556475
EC00344=-1463287,-556475
EC00345=-1463287,-556475
EC00346=-1463287,-556475
EC00347=-1463287,-556475
EC00348=-1463287,-556475
EC00349=-1463287,-556475
EC00350=-1463287,-556475
EC00351=-1463287,-556475
EC00352=-1463287,-556475
EC00353=-1463287,-556475
EC00354=-1463287,-556475
EC00355=-1463287,-556475
EC00356=-1463287,-556475
EC00357=-1463287,-556475
EC00358=-1463287,-556475
EC00359=-1463287,-556475
EC00360=-1463287,-556475
EC00361=-1463287,-556475
EC00362=-1463287,-556475
EC00363=-1463287,-556475
EC00364=-1463287,-556475
EC00365=-1463287,-556475
EC00366=-1463287,-556475
EC00367=-1463287,-556475
EC00368=-1463287,-556475
EC00369=-1463287,-556475
EC00370=-1463287,-556475
EC00371=-1463287,-556475
EC00372=-1463287,-556475
EC00373=-1463287,-556475
EC00374=-1463287,-556475
EC00375=-1463287,-556475
EC00376=-1463287,-556475
EC00377=-1463287,-556475
EC00378=-1463287,-556475
EC00379=-1463287,-556475
EC00380=-1463287,-556475
EC00381=-1463287,-556475
EC00382=-1463287,-556475
EC00383=-1463287,-556475
EC00384=-1463287,-556475
EC00385=-1463287,-556475
EC00386=-1463287,-556475
EC00387=-1463287,-556475
EC00388=-1463287,-556475
EC00389=-1463287,-556475
EC00390=-1463287,-556475
EC00391=-1463287,-556475
EC00392=-1463287,-556475
EC00393=-1463287,-556475
EC00394=-1463287,-556475
EC00395=-1463287,-556475
EC00396=-1463287,-556475
EC00397=-1463287,-556475
EC00398=-1463287,-556475
EC00399=-1463287,-556475
EC00400=-1463287,-556475
EC00401=-1463287,-556475
EC00402=-1463287,-556475
EC00403=-1463287,-556475
EC00404=-1463287,-556475
EC00405=-1463287,-556475
EC00406=-1463287,-556475
EC00407=-1463287,-556475
EC00408=-1463287,-556475
EC00409=-1463287,-556475
EC00410=-1463287,-556475
EC00411=-1463287,-556475
EC00412=-1463287,-556475
EC00413=-1463287,-556475
EC00414=-1463287,-556475
EC00415=-1463287,-556475
EC00416=-1463287,-556475
EC00417=-1463287,-556475
///POSTYPE BASE
///RECTAN
///RCONF 0,0,0,0,0,0,0,0,0,0,0,0,0,0,0,0,0,0,0,0,0,0,0,0
P00006=0.222,-3.123,-1.508,0.0000,0.0000,0.0000
P00021=-0.225,-6.128,-0.405,0.0000,0.0000,0.0000
P00022=0.222,-3.123,-1.508,0.0000,0.0000,0.0000
P00023=0.143,-0.036,0.682,0.0000,0.0000,0.0000
P00024=0.145,-0.552,1.326,0.0000,0.0000,0.0000
P00025=-2.003,0.006,0.728,0.0000,0.0000,0.0000
P00026=0.562,-0.002,-0.337,0.0000,0.0000,0.0000
P00027=-0.746,0.015,-9.096,0.0000,0.0000,0.0000
P00028=-2.237,-0.018,-7.702,0.0000,0.0000,0.0000
P00029=-2.156,-0.086,-4.681,0.0000,0.0000,0.0000
P00030=5.926,-4.294,-1.390,0.0000,0.0000,0.0000
P00031=1.853,-0.001,-1.549,0.0000,0.0000,0.0000
P00032=1.957,0.503,-7.217,0.0000,0.0000,0.0000
///RCONF 0,0,0,0,1,0,0,0,0,0,0,0,0,0,0,0,0,0,0,0,0,0,0,0
P00033=-0.123,0.612,-5.012,0.0000,0.0000,0.0000
///RCONF 0,0,0,0,0,0,0,0,0,0,0,0,0,0,0,0,0,0,0,0,0,0,0,0
P00034=-0.304,0.773,-2.693,0.0000,0.0000,0.0000
P00035=2.817,0.591,-1.622,0.0000,0.0000,0.0000
P00036=-1.108,-0.829,1.850,0.0000,0.0000,0.0000
P00037=0.023,0.937,-2.677,0.0000,0.0000,0.0000
P00038=0.158,-1.133,-1.952,0.0000,0.0000,0.0000
P00039=0.012,-3.081,-0.106,0.0000,0.0000,0.0000
P00040=-0.030,9.648,2.467,0.0000,0.0000,0.0000
//INST
///DATE 2024/02/02 10:05
///ATTR SC,RW
///GROUP1 RB1,BS1
///GROUP2 ST1
NOP
'N_r2_D54(P)(-165,-90)
MOVJ C00000 BC00000 VJ=100.00  +MOVJ EC00000 VJ=100.00
MOVJ C00001 BC00001 VJ=100.00  +MOVJ EC00001 VJ=100.00
MOVJ C00002 BC00002 VJ=100.00  +MOVJ EC00002 VJ=100.00
'Path S3231
SSFTOF
MOVJ C00003 BC00003 VJ=100.00  +MOVJ EC00003 VJ=100.00
MOVL C00004 BC00004 V=400.0  +MOVJ EC00004 VJ=100.00
SMOVL C00005 BC00005 V=60.0  +MOVJ EC00005
SREFP 3 C00006 BC00006  +REFP EC00006
CALL JOB:SEARCH-R1-S1
SET P021 P006
SSFTON P021
SMOVL C00007 BC00007 V=60.0  +MOVJ EC00007
SMOVL C00008 BC00008 V=60.0  +MOVJ EC00008
SREFP 3 C00009 BC00009  +REFP EC00009
CALL JOB:SEARCH-R1-S1
SET P021 P006
SSFTON P021
SMOVL C00010 BC00010 V=60.0  +MOVJ EC00010
MOVL C00011 BC00011 V=400.0  +MOVJ EC00011 VJ=100.00
MOVL C00012 BC00012 V=1000.0  +MOVJ EC00012 VJ=100.00
MOVJ C00013 BC00013 VJ=100.00  +MOVJ EC00013 VJ=100.00
'Path S3232
SSFTOF
MOVJ C00014 BC00014 VJ=100.00  +MOVJ EC00014 VJ=100.00
MOVL C00015 BC00015 V=400.0  +MOVJ EC00015 VJ=100.00
SMOVL C00016 BC00016 V=60.0  +MOVJ EC00016
SREFP 3 C00017 BC00017  +REFP EC00017
CALL JOB:SEARCH-R1-S1
SET P022 P006
SSFTON P022
SMOVL C00018 BC00018 V=60.0  +MOVJ EC00018
SMOVL C00019 BC00019 V=60.0  +MOVJ EC00019
SREFP 3 C00020 BC00020  +REFP EC00020
CALL JOB:SEARCH-R1-S1
SET P022 P006
SSFTON P022
SMOVL C00021 BC00021 V=60.0  +MOVJ EC00021
MOVL C00022 BC00022 V=400.0  +MOVJ EC00022 VJ=100.00
MOVL C00023 BC00023 V=1000.0  +MOVJ EC00023 VJ=100.00
MOVJ C00024 BC00024 VJ=100.00  +MOVJ EC00024 VJ=100.00
'Path S3233
SSFTOF
MOVJ C00025 BC00025 VJ=100.00  +MOVJ EC00025 VJ=100.00
MOVL C00026 BC00026 V=400.0  +MOVJ EC00026 VJ=100.00
SMOVL C00027 BC00027 V=60.0  +MOVJ EC00027
SREFP 3 C00028 BC00028  +REFP EC00028
CALL JOB:SEARCH-R1-S1
SET P023 P006
SSFTON P023
SMOVL C00029 BC00029 V=60.0  +MOVJ EC00029
SMOVL C00030 BC00030 V=60.0  +MOVJ EC00030
SREFP 3 C00031 BC00031  +REFP EC00031
CALL JOB:SEARCH-R1-S1
SET P023 P006
SSFTON P023
SMOVL C00032 BC00032 V=60.0  +MOVJ EC00032
MOVL C00033 BC00033 V=400.0  +MOVJ EC00033 VJ=100.00
MOVL C00034 BC00034 V=1000.0  +MOVJ EC00034 VJ=100.00
MOVJ C00035 BC00035 VJ=100.00  +MOVJ EC00035 VJ=100.00
'Path S3234
SSFTOF
MOVJ C00036 BC00036 VJ=100.00  +MOVJ EC00036 VJ=100.00
MOVL C00037 BC00037 V=400.0  +MOVJ EC00037 VJ=100.00
SMOVL C00038 BC00038 V=60.0  +MOVJ EC00038
SREFP 3 C00039 BC00039  +REFP EC00039
CALL JOB:SEARCH-R1-S1
SET P024 P006
SSFTON P024
SMOVL C00040 BC00040 V=60.0  +MOVJ EC00040
SMOVL C00041 BC00041 V=60.0  +MOVJ EC00041
SREFP 3 C00042 BC00042  +REFP EC00042
CALL JOB:SEARCH-R1-S1
SET P024 P006
SSFTON P024
SMOVL C00043 BC00043 V=60.0  +MOVJ EC00043
MOVL C00044 BC00044 V=400.0  +MOVJ EC00044 VJ=100.00
MOVL C00045 BC00045 V=1000.0  +MOVJ EC00045 VJ=100.00
MOVJ C00046 BC00046 VJ=100.00  +MOVJ EC00046 VJ=100.00
'Path S3235
SSFTOF
MOVJ C00047 BC00047 VJ=100.00  +MOVJ EC00047 VJ=100.00
MOVL C00048 BC00048 V=400.0  +MOVJ EC00048 VJ=100.00
SMOVL C00049 BC00049 V=60.0  +MOVJ EC00049
SREFP 3 C00050 BC00050  +REFP EC00050
CALL JOB:SEARCH-R1-S1
SET P025 P006
SSFTON P025
SMOVL C00051 BC00051 V=60.0  +MOVJ EC00051
SMOVL C00052 BC00052 V=60.0  +MOVJ EC00052
SREFP 3 C00053 BC00053  +REFP EC00053
CALL JOB:SEARCH-R1-S1
SET P025 P006
SSFTON P025
SMOVL C00054 BC00054 V=60.0  +MOVJ EC00054
MOVL C00055 BC00055 V=400.0  +MOVJ EC00055 VJ=100.00
MOVL C00056 BC00056 V=1000.0  +MOVJ EC00056 VJ=100.00
MOVJ C00057 BC00057 VJ=100.00  +MOVJ EC00057 VJ=100.00
'Path S3236
SSFTOF
MOVJ C00058 BC00058 VJ=100.00  +MOVJ EC00058 VJ=100.00
MOVL C00059 BC00059 V=400.0  +MOVJ EC00059 VJ=100.00
SMOVL C00060 BC00060 V=60.0  +MOVJ EC00060
SREFP 3 C00061 BC00061  +REFP EC00061
CALL JOB:SEARCH-R1-S1
SET P026 P006
SSFTON P026
SMOVL C00062 BC00062 V=60.0  +MOVJ EC00062
SMOVL C00063 BC00063 V=60.0  +MOVJ EC00063
SREFP 3 C00064 BC00064  +REFP EC00064
CALL JOB:SEARCH-R1-S1
SET P026 P006
SSFTON P026
SMOVL C00065 BC00065 V=60.0  +MOVJ EC00065
MOVL C00066 BC00066 V=400.0  +MOVJ EC00066 VJ=100.00
MOVL C00067 BC00067 V=1000.0  +MOVJ EC00067 VJ=100.00
'obrot
MOVJ C00068 BC00068 VJ=100.00  +MOVJ EC00068 VJ=100.00
MOVJ C00069 BC00069 VJ=100.00  +MOVJ EC00069 VJ=100.00
MOVJ C00070 BC00070 VJ=100.00  +MOVJ EC00070 VJ=100.00
MOVJ C00071 BC00071 VJ=100.00  +MOVJ EC00071 VJ=100.00
MOVJ C00072 BC00072 VJ=100.00  +MOVJ EC00072 VJ=100.00
MOVJ C00073 BC00073 VJ=100.00  +MOVJ EC00073 VJ=100.00
'Path S3270
SSFTOF
MOVJ C00074 BC00074 VJ=100.00  +MOVJ EC00074 VJ=100.00
MOVL C00075 BC00075 V=400.0  +MOVJ EC00075 VJ=100.00
SMOVL C00076 BC00076 V=100.0  +MOVJ EC00076
SREFP 3 C00077 BC00077  +REFP EC00077
CALL JOB:SEARCH-R1-S1
SET P027 P006
SSFTON P027
SMOVL C00078 BC00078 V=100.0  +MOVJ EC00078
SMOVL C00079 BC00079 V=100.0  +MOVJ EC00079
SREFP 3 C00080 BC00080  +REFP EC00080
CALL JOB:SEARCH-R1-S1
SET P027 P006
SSFTON P027
SMOVL C00081 BC00081 V=100.0  +MOVJ EC00081
MOVL C00082 BC00082 V=400.0  +MOVJ EC00082 VJ=100.00
MOVL C00083 BC00083 V=1000.0  +MOVJ EC00083 VJ=100.00
'Path S3271
SSFTOF
MOVJ C00084 BC00084 VJ=100.00  +MOVJ EC00084 VJ=100.00
MOVL C00085 BC00085 V=400.0  +MOVJ EC00085 VJ=100.00
SMOVL C00086 BC00086 V=100.0  +MOVJ EC00086
SREFP 3 C00087 BC00087  +REFP EC00087
CALL JOB:SEARCH-R1-S1
SET P028 P006
SSFTON P028
SMOVL C00088 BC00088 V=100.0  +MOVJ EC00088
SMOVL C00089 BC00089 V=100.0  +MOVJ EC00089
SREFP 3 C00090 BC00090  +REFP EC00090
CALL JOB:SEARCH-R1-S1
SET P028 P006
SSFTON P028
SMOVL C00091 BC00091 V=100.0  +MOVJ EC00091
MOVL C00092 BC00092 V=400.0  +MOVJ EC00092 VJ=100.00
MOVL C00093 BC00093 V=1000.0  +MOVJ EC00093 VJ=100.00
MOVJ C00094 BC00094 VJ=100.00  +MOVJ EC00094 VJ=100.00
'Path S3271
SSFTOF
MOVJ C00095 BC00095 VJ=100.00  +MOVJ EC00095 VJ=100.00
MOVL C00096 BC00096 V=400.0  +MOVJ EC00096 VJ=100.00
SMOVL C00097 BC00097 V=100.0  +MOVJ EC00097
SREFP 3 C00098 BC00098  +REFP EC00098
CALL JOB:SEARCH-R1-S1
SET P029 P006
SSFTON P029
SMOVL C00099 BC00099 V=100.0  +MOVJ EC00099
SMOVL C00100 BC00100 V=100.0  +MOVJ EC00100
SREFP 3 C00101 BC00101  +REFP EC00101
CALL JOB:SEARCH-R1-S1
SET P029 P006
SSFTON P029
SMOVL C00102 BC00102 V=100.0  +MOVJ EC00102
MOVL C00103 BC00103 V=400.0  +MOVJ EC00103 VJ=100.00
MOVL C00104 BC00104 V=1000.0  +MOVJ EC00104 VJ=100.00
'Path S3272
SSFTOF
MOVJ C00105 BC00105 VJ=100.00  +MOVJ EC00105 VJ=100.00
MOVL C00106 BC00106 V=400.0  +MOVJ EC00106 VJ=100.00
SMOVL C00107 BC00107 V=100.0  +MOVJ EC00107
SREFP 3 C00108 BC00108  +REFP EC00108
CALL JOB:SEARCH-R1-S1
SET P030 P006
SSFTON P030
SMOVL C00109 BC00109 V=100.0  +MOVJ EC00109
SMOVL C00110 BC00110 V=100.0  +MOVJ EC00110
SREFP 3 C00111 BC00111  +REFP EC00111
CALL JOB:SEARCH-R1-S1
SET P030 P006
SSFTON P030
SMOVL C00112 BC00112 V=100.0  +MOVJ EC00112
MOVL C00113 BC00113 V=400.0  +MOVJ EC00113 VJ=100.00
MOVL C00114 BC00114 V=1000.0  +MOVJ EC00114 VJ=100.00
MOVJ C00115 BC00115 VJ=100.00  +MOVJ EC00115 VJ=100.00
MOVJ C00116 BC00116 VJ=100.00  +MOVJ EC00116 VJ=100.00
MOVJ C00117 BC00117 VJ=100.00  +MOVJ EC00117 VJ=100.00
'
MOVJ C00118 BC00118 VJ=100.00  +MOVJ EC00118 VJ=100.00
MOVJ C00119 BC00119 VJ=100.00  +MOVJ EC00119 VJ=100.00
MOVJ C00120 BC00120 VJ=100.00  +MOVJ EC00120 VJ=100.00
MOVJ C00121 BC00121 VJ=100.00  +MOVJ EC00121 VJ=100.00
MOVJ C00122 BC00122 VJ=100.00  +MOVJ EC00122 VJ=100.00
MOVJ C00123 BC00123 VJ=100.00  +MOVJ EC00123 VJ=100.00
'Path S3272
SSFTOF
MOVJ C00124 BC00124 VJ=100.00  +MOVJ EC00124 VJ=100.00
MOVL C00125 BC00125 V=400.0  +MOVJ EC00125 VJ=100.00
SMOVL C00126 BC00126 V=100.0  +MOVJ EC00126
SREFP 3 C00127 BC00127  +REFP EC00127
CALL JOB:SEARCH-R1-S1
SET P037 P006
SSFTON P037
SMOVL C00128 BC00128 V=100.0  +MOVJ EC00128
SMOVL C00129 BC00129 V=100.0  +MOVJ EC00129
SREFP 3 C00130 BC00130  +REFP EC00130
CALL JOB:SEARCH-R1-S1
SET P037 P006
SSFTON P037
SMOVL C00131 BC00131 V=100.0  +MOVJ EC00131
SMOVL C00132 BC00132 V=100.0  +MOVJ EC00132
SREFP 3 C00133 BC00133  +REFP EC00133
CALL JOB:SEARCH-R1-S1
SET P037 P006
SSFTON P037
SMOVL C00134 BC00134 V=100.0  +MOVJ EC00134
MOVL C00135 BC00135 V=400.0  +MOVJ EC00135 VJ=100.00
MOVL C00136 BC00136 V=1000.0  +MOVJ EC00136 VJ=100.00
'Path S3273
SSFTOF
MOVJ C00137 BC00137 VJ=100.00  +MOVJ EC00137 VJ=100.00
MOVL C00138 BC00138 V=400.0  +MOVJ EC00138 VJ=100.00
SMOVL C00139 BC00139 V=100.0  +MOVJ EC00139
SREFP 3 C00140 BC00140  +REFP EC00140
CALL JOB:SEARCH-R1-S1
SET P038 P006
SSFTON P038
SMOVL C00141 BC00141 V=100.0  +MOVJ EC00141
SMOVL C00142 BC00142 V=100.0  +MOVJ EC00142
SREFP 3 C00143 BC00143  +REFP EC00143
CALL JOB:SEARCH-R1-S1
SET P038 P006
SSFTON P038
SMOVL C00144 BC00144 V=100.0  +MOVJ EC00144
MOVL C00145 BC00145 V=400.0  +MOVJ EC00145 VJ=100.00
MOVL C00146 BC00146 V=1000.0  +MOVJ EC00146 VJ=100.00
MOVJ C00147 BC00147 VJ=100.00  +MOVJ EC00147 VJ=100.00
'Path S3273
SSFTOF
MOVJ C00148 BC00148 VJ=100.00  +MOVJ EC00148 VJ=100.00
MOVL C00149 BC00149 V=400.0  +MOVJ EC00149 VJ=100.00
SMOVL C00150 BC00150 V=100.0  +MOVJ EC00150
SREFP 3 C00151 BC00151  +REFP EC00151
CALL JOB:SEARCH-R1-S1
SET P039 P006
SSFTON P039
SMOVL C00152 BC00152 V=100.0  +MOVJ EC00152
SMOVL C00153 BC00153 V=100.0  +MOVJ EC00153
SREFP 3 C00154 BC00154  +REFP EC00154
CALL JOB:SEARCH-R1-S1
SET P039 P006
SSFTON P039
SMOVL C00155 BC00155 V=100.0  +MOVJ EC00155
MOVL C00156 BC00156 V=400.0  +MOVJ EC00156 VJ=100.00
MOVL C00157 BC00157 V=1000.0  +MOVJ EC00157 VJ=100.00
'Path S3274
SSFTOF
MOVJ C00158 BC00158 VJ=100.00  +MOVJ EC00158 VJ=100.00
MOVL C00159 BC00159 V=400.0  +MOVJ EC00159 VJ=100.00
SMOVL C00160 BC00160 V=100.0  +MOVJ EC00160
SREFP 3 C00161 BC00161  +REFP EC00161
CALL JOB:SEARCH-R1-S1
SET P040 P006
SSFTON P040
SMOVL C00162 BC00162 V=100.0  +MOVJ EC00162
SMOVL C00163 BC00163 V=100.0  +MOVJ EC00163
SREFP 3 C00164 BC00164  +REFP EC00164
CALL JOB:SEARCH-R1-S1
SET P040 P006
SSFTON P040
SMOVL C00165 BC00165 V=100.0  +MOVJ EC00165
MOVL C00166 BC00166 V=400.0  +MOVJ EC00166 VJ=100.00
MOVL C00167 BC00167 V=1000.0  +MOVJ EC00167 VJ=100.00
MOVJ C00168 BC00168 VJ=100.00  +MOVJ EC00168 VJ=100.00
MOVJ C00169 BC00169 VJ=100.00  +MOVJ EC00169 VJ=100.00
MOVJ C00170 BC00170 VJ=100.00  +MOVJ EC00170 VJ=100.00
MOVJ C00171 BC00171 VJ=100.00  +MOVJ EC00171 VJ=100.00
MOVJ C00172 BC00172 VJ=100.00  +MOVJ EC00172 VJ=100.00
'
'Path S3274
SSFTOF
MOVJ C00173 BC00173 VJ=100.00  +MOVJ EC00173 VJ=100.00
MOVL C00174 BC00174 V=400.0  +MOVJ EC00174 VJ=100.00
SMOVL C00175 BC00175 V=60.0  +MOVJ EC00175
SREFP 3 C00176 BC00176  +REFP EC00176
CALL JOB:SEARCH-R1-S1
SET P034 P006
SSFTON P034
SMOVL C00177 BC00177 V=60.0  +MOVJ EC00177
SMOVL C00178 BC00178 V=60.0  +MOVJ EC00178
SREFP 3 C00179 BC00179  +REFP EC00179
CALL JOB:SEARCH-R1-S1
SET P034 P006
SSFTON P034
SMOVL C00180 BC00180 V=60.0  +MOVJ EC00180
MOVL C00181 BC00181 V=400.0  +MOVJ EC00181 VJ=100.00
MOVL C00182 BC00182 V=1000.0  +MOVJ EC00182 VJ=100.00
'Path S3275
SSFTOF
MOVJ C00183 BC00183 VJ=100.00  +MOVJ EC00183 VJ=100.00
MOVL C00184 BC00184 V=400.0  +MOVJ EC00184 VJ=100.00
SMOVL C00185 BC00185 V=60.0  +MOVJ EC00185
SREFP 3 C00186 BC00186  +REFP EC00186
CALL JOB:SEARCH-R1-S1
SET P035 P006
SSFTON P035
SMOVL C00187 BC00187 V=60.0  +MOVJ EC00187
SMOVL C00188 BC00188 V=60.0  +MOVJ EC00188
SREFP 3 C00189 BC00189  +REFP EC00189
CALL JOB:SEARCH-R1-S1
SET P035 P006
SSFTON P035
SMOVL C00190 BC00190 V=60.0  +MOVJ EC00190
MOVL C00191 BC00191 V=400.0  +MOVJ EC00191 VJ=100.00
MOVL C00192 BC00192 V=1000.0  +MOVJ EC00192 VJ=100.00
MOVJ C00193 BC00193 VJ=100.00  +MOVJ EC00193 VJ=100.00
'Path S3276
SSFTOF
MOVJ C00194 BC00194 VJ=100.00  +MOVJ EC00194 VJ=100.00
MOVL C00195 BC00195 V=400.0  +MOVJ EC00195 VJ=100.00
SMOVL C00196 BC00196 V=60.0  +MOVJ EC00196
SREFP 3 C00197 BC00197  +REFP EC00197
CALL JOB:SEARCH-R1-S1
SET P036 P006
SSFTON P036
SMOVL C00198 BC00198 V=60.0  +MOVJ EC00198
SMOVL C00199 BC00199 V=60.0  +MOVJ EC00199
SREFP 3 C00200 BC00200  +REFP EC00200
CALL JOB:SEARCH-R1-S1
SET P036 P006
SSFTON P036
SMOVL C00201 BC00201 V=60.0  +MOVJ EC00201
MOVL C00202 BC00202 V=400.0  +MOVJ EC00202 VJ=100.00
MOVL C00203 BC00203 V=1000.0  +MOVJ EC00203 VJ=100.00
'Path S3277
SSFTOF
MOVJ C00204 BC00204 VJ=100.00  +MOVJ EC00204 VJ=100.00
MOVL C00205 BC00205 V=400.0  +MOVJ EC00205 VJ=100.00
SMOVL C00206 BC00206 V=60.0  +MOVJ EC00206
SREFP 3 C00207 BC00207  +REFP EC00207
CALL JOB:SEARCH-R1-S1
SET P031 P006
SSFTON P031
SMOVL C00208 BC00208 V=60.0  +MOVJ EC00208
SMOVL C00209 BC00209 V=60.0  +MOVJ EC00209
SREFP 3 C00210 BC00210  +REFP EC00210
CALL JOB:SEARCH-R1-S1
SET P031 P006
SSFTON P031
SMOVL C00211 BC00211 V=60.0  +MOVJ EC00211
MOVL C00212 BC00212 V=400.0  +MOVJ EC00212 VJ=100.00
MOVL C00213 BC00213 V=1000.0  +MOVJ EC00213 VJ=100.00
MOVJ C00214 BC00214 VJ=100.00  +MOVJ EC00214 VJ=100.00
'Path S3278
SSFTOF
MOVJ C00215 BC00215 VJ=100.00  +MOVJ EC00215 VJ=100.00
MOVL C00216 BC00216 V=400.0  +MOVJ EC00216 VJ=100.00
SMOVL C00217 BC00217 V=60.0  +MOVJ EC00217
SREFP 3 C00218 BC00218  +REFP EC00218
CALL JOB:SEARCH-R1-S1
SET P032 P006
SSFTON P032
SMOVL C00219 BC00219 V=60.0  +MOVJ EC00219
SMOVL C00220 BC00220 V=60.0  +MOVJ EC00220
SREFP 3 C00221 BC00221  +REFP EC00221
CALL JOB:SEARCH-R1-S1
SET P032 P006
SSFTON P032
SMOVL C00222 BC00222 V=60.0  +MOVJ EC00222
MOVL C00223 BC00223 V=400.0  +MOVJ EC00223 VJ=100.00
MOVL C00224 BC00224 V=1000.0  +MOVJ EC00224 VJ=100.00
'Path S3279
SSFTOF
MOVJ C00225 BC00225 VJ=100.00  +MOVJ EC00225 VJ=100.00
MOVL C00226 BC00226 V=400.0  +MOVJ EC00226 VJ=100.00
SMOVL C00227 BC00227 V=60.0  +MOVJ EC00227
SREFP 3 C00228 BC00228  +REFP EC00228
CALL JOB:SEARCH-R1-S1
SET P033 P006
SSFTON P033
SMOVL C00229 BC00229 V=60.0  +MOVJ EC00229
SMOVL C00230 BC00230 V=60.0  +MOVJ EC00230
SREFP 3 C00231 BC00231  +REFP EC00231
CALL JOB:SEARCH-R1-S1
SET P033 P006
SSFTON P033
SMOVL C00232 BC00232 V=60.0  +MOVJ EC00232
MOVL C00233 BC00233 V=400.0  +MOVJ EC00233 VJ=100.00
MOVL C00234 BC00234 V=1000.0  +MOVJ EC00234 VJ=100.00
'
MOVJ C00235 BC00235 VJ=100.00  +MOVJ EC00235 VJ=100.00
MOVJ C00236 BC00236 VJ=100.00  +MOVJ EC00236 VJ=100.00
'
'
'Path W3280
SSFTOF
SSFTON P034
MOVJ C00237 BC00237 VJ=100.00  +MOVJ EC00237 VJ=100.00
SMOVL C00238 BC00238 V=400.0  +MOVJ EC00238
SMOVL C00239 BC00239 V=100.0 PL=0  +MOVJ EC00239
SREFP 1 C00240 BC00240  +REFP EC00240
SREFP 2 C00241 BC00241  +REFP EC00241
MACRO1 MJ#(0) ARGF0
ARCON
SMOVL C00242 BC00242 V=10.0  +MOVJ EC00242
SMOVL C00243 BC00243 V=10.0  +MOVJ EC00243
SMOVL C00244 BC00244 V=10.0  +MOVJ EC00244
ARCOF
SMOVL C00245 BC00245 V=400.0  +MOVJ EC00245
SMOVL C00246 BC00246 V=1000.0  +MOVJ EC00246
SSFTOF
'Path W3281
SSFTOF
SSFTON P035
MOVJ C00247 BC00247 VJ=100.00  +MOVJ EC00247 VJ=100.00
SMOVL C00248 BC00248 V=400.0  +MOVJ EC00248
SMOVL C00249 BC00249 V=100.0 PL=0  +MOVJ EC00249
SREFP 1 C00250 BC00250  +REFP EC00250
SREFP 2 C00251 BC00251  +REFP EC00251
MACRO1 MJ#(0) ARGF0
ARCON
SMOVL C00252 BC00252 V=10.0  +MOVJ EC00252
SMOVL C00253 BC00253 V=10.0  +MOVJ EC00253
SMOVL C00254 BC00254 V=10.0  +MOVJ EC00254
ARCOF
SMOVL C00255 BC00255 V=400.0  +MOVJ EC00255
SMOVL C00256 BC00256 V=1000.0  +MOVJ EC00256
SSFTOF
MOVJ C00257 BC00257 VJ=100.00  +MOVJ EC00257 VJ=100.00
'Path W3282
SSFTOF
SSFTON P036
MOVJ C00258 BC00258 VJ=100.00  +MOVJ EC00258 VJ=100.00
SMOVL C00259 BC00259 V=400.0  +MOVJ EC00259
SMOVL C00260 BC00260 V=100.0 PL=0  +MOVJ EC00260
SREFP 1 C00261 BC00261  +REFP EC00261
SREFP 2 C00262 BC00262  +REFP EC00262
MACRO1 MJ#(0) ARGF0
ARCON
SMOVL C00263 BC00263 V=10.0  +MOVJ EC00263
SMOVL C00264 BC00264 V=10.0  +MOVJ EC00264
SMOVL C00265 BC00265 V=10.0  +MOVJ EC00265
ARCOF
SMOVL C00266 BC00266 V=400.0  +MOVJ EC00266
SMOVL C00267 BC00267 V=1000.0  +MOVJ EC00267
SSFTOF
'Path W3283
SSFTOF
SSFTON P031
MOVJ C00268 BC00268 VJ=100.00  +MOVJ EC00268 VJ=100.00
SMOVL C00269 BC00269 V=400.0  +MOVJ EC00269
SMOVL C00270 BC00270 V=100.0 PL=0  +MOVJ EC00270
SREFP 1 C00271 BC00271  +REFP EC00271
SREFP 2 C00272 BC00272  +REFP EC00272
MACRO1 MJ#(0) ARGF0
ARCON
SMOVL C00273 BC00273 V=10.0  +MOVJ EC00273
SMOVL C00274 BC00274 V=10.0  +MOVJ EC00274
SMOVL C00275 BC00275 V=10.0  +MOVJ EC00275
ARCOF
SMOVL C00276 BC00276 V=400.0  +MOVJ EC00276
SMOVL C00277 BC00277 V=1000.0  +MOVJ EC00277
SSFTOF
MOVJ C00278 BC00278 VJ=100.00  +MOVJ EC00278 VJ=100.00
'Path W3284
SSFTOF
SSFTON P032
MOVJ C00279 BC00279 VJ=100.00  +MOVJ EC00279 VJ=100.00
SMOVL C00280 BC00280 V=400.0  +MOVJ EC00280
SMOVL C00281 BC00281 V=100.0 PL=0  +MOVJ EC00281
SREFP 1 C00282 BC00282  +REFP EC00282
SREFP 2 C00283 BC00283  +REFP EC00283
MACRO1 MJ#(0) ARGF0
ARCON
SMOVL C00284 BC00284 V=10.0  +MOVJ EC00284
SMOVL C00285 BC00285 V=10.0  +MOVJ EC00285
SMOVL C00286 BC00286 V=10.0  +MOVJ EC00286
ARCOF
SMOVL C00287 BC00287 V=400.0  +MOVJ EC00287
SMOVL C00288 BC00288 V=1000.0  +MOVJ EC00288
SSFTOF
'Path W3285
SSFTOF
SSFTON P033
MOVJ C00289 BC00289 VJ=100.00  +MOVJ EC00289 VJ=100.00
SMOVL C00290 BC00290 V=400.0  +MOVJ EC00290
SMOVL C00291 BC00291 V=100.0 PL=0  +MOVJ EC00291
SREFP 1 C00292 BC00292  +REFP EC00292
SREFP 2 C00293 BC00293  +REFP EC00293
MACRO1 MJ#(0) ARGF0
ARCON
SMOVL C00294 BC00294 V=10.0  +MOVJ EC00294
SMOVL C00295 BC00295 V=10.0  +MOVJ EC00295
SMOVL C00296 BC00296 V=10.0  +MOVJ EC00296
ARCOF
SMOVL C00297 BC00297 V=400.0  +MOVJ EC00297
SMOVL C00298 BC00298 V=1000.0  +MOVJ EC00298
SSFTOF
'obrot
MOVJ C00299 BC00299 VJ=100.00  +MOVJ EC00299 VJ=100.00
MOVJ C00300 BC00300 VJ=100.00  +MOVJ EC00300 VJ=100.00
MOVJ C00301 BC00301 VJ=100.00  +MOVJ EC00301 VJ=100.00
MOVJ C00302 BC00302 VJ=100.00  +MOVJ EC00302 VJ=100.00
'Path W3267
SSFTOF
SSFTON P040
MOVJ C00303 BC00303 VJ=100.00  +MOVJ EC00303 VJ=100.00
SMOVL C00304 BC00304 V=400.0  +MOVJ EC00304
SMOVL C00305 BC00305 V=100.0 PL=0  +MOVJ EC00305
SREFP 1 C00306 BC00306  +REFP EC00306
SREFP 2 C00307 BC00307  +REFP EC00307
MACRO1 MJ#(0) ARGF0
ARCON
SSFTON P039
SMOVL C00308 BC00308 V=10.0  +MOVJ EC00308
ARCOF
SMOVL C00309 BC00309 V=400.0  +MOVJ EC00309
SMOVL C00310 BC00310 V=1000.0  +MOVJ EC00310
SSFTOF
MOVJ C00311 BC00311 VJ=100.00  +MOVJ EC00311 VJ=100.00
'Path W3269
SSFTOF
SSFTON P038
MOVJ C00312 BC00312 VJ=100.00  +MOVJ EC00312 VJ=100.00
SMOVL C00313 BC00313 V=400.0  +MOVJ EC00313
SMOVL C00314 BC00314 V=150.0 PL=0  +MOVJ EC00314
SREFP 1 C00315 BC00315  +REFP EC00315
SREFP 2 C00316 BC00316  +REFP EC00316
MACRO1 MJ#(0) ARGF0
ARCON
SMOVL C00317 BC00317 V=10.0  +MOVJ EC00317
SSFTON P037
SMOVL C00318 BC00318 V=10.0  +MOVJ EC00318
ARCOF
SMOVL C00319 BC00319 V=400.0  +MOVJ EC00319
SMOVL C00320 BC00320 V=1000.0  +MOVJ EC00320
SSFTOF
MOVJ C00321 BC00321 VJ=100.00  +MOVJ EC00321 VJ=100.00
MOVJ C00322 BC00322 VJ=100.00  +MOVJ EC00322 VJ=100.00
MOVJ C00323 BC00323 VJ=100.00  +MOVJ EC00323 VJ=100.00
MOVJ C00324 BC00324 VJ=100.00  +MOVJ EC00324 VJ=100.00
MOVJ C00325 BC00325 VJ=100.00  +MOVJ EC00325 VJ=100.00
MOVJ C00326 BC00326 VJ=100.00  +MOVJ EC00326 VJ=100.00
MOVJ C00327 BC00327 VJ=100.00  +MOVJ EC00327 VJ=100.00
MOVJ C00328 BC00328 VJ=100.00  +MOVJ EC00328 VJ=100.00
MOVJ C00329 BC00329 VJ=100.00  +MOVJ EC00329 VJ=100.00
'
'Path W3286
SSFTOF
SSFTON P021
MOVJ C00330 BC00330 VJ=100.00  +MOVJ EC00330 VJ=100.00
SMOVL C00331 BC00331 V=400.0  +MOVJ EC00331
SMOVL C00332 BC00332 V=100.0 PL=0  +MOVJ EC00332
SREFP 1 C00333 BC00333  +REFP EC00333
SREFP 2 C00334 BC00334  +REFP EC00334
MACRO1 MJ#(0) ARGF0
ARCON
SMOVL C00335 BC00335 V=10.0  +MOVJ EC00335
SMOVL C00336 BC00336 V=10.0  +MOVJ EC00336
SMOVL C00337 BC00337 V=10.0  +MOVJ EC00337
ARCOF
SMOVL C00338 BC00338 V=400.0  +MOVJ EC00338
SMOVL C00339 BC00339 V=1000.0  +MOVJ EC00339
SSFTOF
MOVJ C00340 BC00340 VJ=100.00  +MOVJ EC00340 VJ=100.00
'Path W3287
SSFTOF
SSFTON P022
MOVJ C00341 BC00341 VJ=100.00  +MOVJ EC00341 VJ=100.00
SMOVL C00342 BC00342 V=400.0  +MOVJ EC00342
SMOVL C00343 BC00343 V=100.0 PL=0  +MOVJ EC00343
SREFP 1 C00344 BC00344  +REFP EC00344
SREFP 2 C00345 BC00345  +REFP EC00345
MACRO1 MJ#(0) ARGF0
ARCON
SMOVL C00346 BC00346 V=10.0  +MOVJ EC00346
SMOVL C00347 BC00347 V=10.0  +MOVJ EC00347
SMOVL C00348 BC00348 V=10.0  +MOVJ EC00348
ARCOF
SMOVL C00349 BC00349 V=400.0  +MOVJ EC00349
SMOVL C00350 BC00350 V=1000.0  +MOVJ EC00350
SSFTOF
MOVJ C00351 BC00351 VJ=100.00  +MOVJ EC00351 VJ=100.00
'Path W3288
SSFTOF
SSFTON P023
MOVJ C00352 BC00352 VJ=100.00  +MOVJ EC00352 VJ=100.00
SMOVL C00353 BC00353 V=400.0  +MOVJ EC00353
SMOVL C00354 BC00354 V=100.0 PL=0  +MOVJ EC00354
SREFP 1 C00355 BC00355  +REFP EC00355
SREFP 2 C00356 BC00356  +REFP EC00356
MACRO1 MJ#(0) ARGF0
ARCON
SMOVL C00357 BC00357 V=10.0  +MOVJ EC00357
SMOVL C00358 BC00358 V=10.0  +MOVJ EC00358
SMOVL C00359 BC00359 V=10.0  +MOVJ EC00359
ARCOF
SMOVL C00360 BC00360 V=400.0  +MOVJ EC00360
SMOVL C00361 BC00361 V=1000.0  +MOVJ EC00361
SSFTOF
MOVJ C00362 BC00362 VJ=100.00  +MOVJ EC00362 VJ=100.00
'Path W3289
SSFTOF
SSFTON P023
MOVJ C00363 BC00363 VJ=100.00  +MOVJ EC00363 VJ=100.00
SMOVL C00364 BC00364 V=400.0  +MOVJ EC00364
SMOVL C00365 BC00365 V=100.0 PL=0  +MOVJ EC00365
SREFP 1 C00366 BC00366  +REFP EC00366
SREFP 2 C00367 BC00367  +REFP EC00367
MACRO1 MJ#(0) ARGF0
ARCON
SMOVL C00368 BC00368 V=10.0  +MOVJ EC00368
SMOVL C00369 BC00369 V=10.0  +MOVJ EC00369
SMOVL C00370 BC00370 V=10.0  +MOVJ EC00370
ARCOF
SMOVL C00371 BC00371 V=400.0  +MOVJ EC00371
SMOVL C00372 BC00372 V=1000.0  +MOVJ EC00372
SSFTOF
MOVJ C00373 BC00373 VJ=100.00  +MOVJ EC00373 VJ=100.00
'Path W3290
SSFTOF
SSFTON P022
MOVJ C00374 BC00374 VJ=100.00  +MOVJ EC00374 VJ=100.00
SMOVL C00375 BC00375 V=400.0  +MOVJ EC00375
SMOVL C00376 BC00376 V=100.0 PL=0  +MOVJ EC00376
SREFP 1 C00377 BC00377  +REFP EC00377
SREFP 2 C00378 BC00378  +REFP EC00378
MACRO1 MJ#(0) ARGF0
ARCON
SMOVL C00379 BC00379 V=10.0  +MOVJ EC00379
SMOVL C00380 BC00380 V=10.0  +MOVJ EC00380
SMOVL C00381 BC00381 V=10.0  +MOVJ EC00381
ARCOF
SMOVL C00382 BC00382 V=400.0  +MOVJ EC00382
SMOVL C00383 BC00383 V=1000.0  +MOVJ EC00383
SSFTOF
MOVJ C00384 BC00384 VJ=100.00  +MOVJ EC00384 VJ=100.00
'Path W3291
SSFTOF
SSFTON P021
MOVJ C00385 BC00385 VJ=100.00  +MOVJ EC00385 VJ=100.00
SMOVL C00386 BC00386 V=400.0  +MOVJ EC00386
SMOVL C00387 BC00387 V=100.0 PL=0  +MOVJ EC00387
SREFP 1 C00388 BC00388  +REFP EC00388
SREFP 2 C00389 BC00389  +REFP EC00389
MACRO1 MJ#(0) ARGF0
ARCON
SMOVL C00390 BC00390 V=10.0  +MOVJ EC00390
SMOVL C00391 BC00391 V=10.0  +MOVJ EC00391
SMOVL C00392 BC00392 V=10.0  +MOVJ EC00392
ARCOF
SMOVL C00393 BC00393 V=400.0  +MOVJ EC00393
SMOVL C00394 BC00394 V=1000.0  +MOVJ EC00394
SSFTOF
MOVJ C00395 BC00395 VJ=100.00  +MOVJ EC00395 VJ=100.00
MOVJ C00396 BC00396 VJ=100.00  +MOVJ EC00396 VJ=100.00
MOVJ C00397 BC00397 VJ=100.00  +MOVJ EC00397 VJ=100.00
MOVJ C00398 BC00398 VJ=100.00  +MOVJ EC00398 VJ=100.00
'Path W3262
SSFTOF
SSFTON P028
MOVJ C00399 BC00399 VJ=100.00  +MOVJ EC00399 VJ=100.00
SMOVL C00400 BC00400 V=400.0  +MOVJ EC00400
SMOVL C00401 BC00401 V=100.0 PL=0  +MOVJ EC00401
SREFP 1 C00402 BC00402  +REFP EC00402
SREFP 2 C00403 BC00403  +REFP EC00403
MACRO1 MJ#(0) ARGF0
ARCON
SSFTON P027
SMOVL C00404 BC00404 V=10.0  +MOVJ EC00404
ARCOF
SMOVL C00405 BC00405 V=400.0  +MOVJ EC00405
SMOVL C00406 BC00406 V=1000.0  +MOVJ EC00406
SSFTOF
MOVJ C00407 BC00407 VJ=100.00  +MOVJ EC00407 VJ=100.00
'Path W3264
SSFTOF
SSFTON P030
MOVJ C00408 BC00408 VJ=100.00  +MOVJ EC00408 VJ=100.00
SMOVL C00409 BC00409 V=400.0  +MOVJ EC00409
SMOVL C00410 BC00410 V=100.0 PL=0  +MOVJ EC00410
SREFP 1 C00411 BC00411  +REFP EC00411
SREFP 2 C00412 BC00412  +REFP EC00412
MACRO1 MJ#(0) ARGF0
ARCON
SSFTON P029
SMOVL C00413 BC00413 V=10.0  +MOVJ EC00413
ARCOF
SMOVL C00414 BC00414 V=400.0  +MOVJ EC00414
SMOVL C00415 BC00415 V=1000.0  +MOVJ EC00415
SSFTOF
MOVJ C00416 BC00416 VJ=100.00  +MOVJ EC00416 VJ=100.00
MOVJ C00417 BC00417 VJ=100.00  +MOVJ EC00417 VJ=100.00
END
